(* IEC 61131-3 sources: Industry-PLC-LLM/data/PLCBEAD_repo/PLCBEAD_PLCEmbed-main/PLC-BEAD/Source/GEB/SPHERE_V, 1 file *)

(* ---- SPHERE_V.ST ---- *)
FUNCTION SPHERE_V:REAL

	VAR_INPUT
		RX :	REAL;
	END_VAR

	sphere_V := 4.188790205 * RX * RX * RX;

END_FUNCTION

PROGRAM program0

	VAR
		RX :	REAL;
		CEIL5_OUT : REAL;
	END_VAR

	CEIL5_OUT := SPHERE_V(RX);

END_PROGRAM
